// TIA Portal V19 export
DATA_BLOCK "GetPrg_DB"   // DB83
// stored: InstanceOfName GetPrg, InstanceOfType FB
"GetPrg"
   // VAR_INPUT
   //    Execute : Bool;
   //    PrgNo : DInt;
   // END_VAR
   // VAR_OUTPUT
   //    Busy : Bool;
   //    Done : Bool;
   //    Error : Bool;
   //    workTime : LTime;
   // END_VAR
   // VAR_IN_OUT
   //    GET_ITF : "Prg_GetITF";
   //    GET_Data : Variant;
   //    PRG_Data : Variant;
   // END_VAR
   // VAR
   //    Status : Int;
   //    iTime { S7_SetPoint := 'True'} : DTL;
   // END_VAR
BEGIN
END_DATA_BLOCK
